(* Logix 5000 project; controller EDS_V35 1769-L16ER-BB1B rev 35.11; software revision 35.00 *)

TASK MainTask (continuous, watchdog 500 ms) : MainProgram

MODULES
   Local : 1769-L16ER-BB1B (PointIO 0, rev 35.11)
      G2410 : vendor 1256 type 43 code 1 (Ethernet 192.168.1.17, rev 6.3, StandardDataDriven RPI 10 ms)
      Discrete_IO : Embedded (PointIO 1, rev 35.11, Output RPI 20 ms)
END_MODULES

PROGRAM MainProgram   (* main routine MainRoutine *)

ROUTINE MainRoutine   (* ladder *)
END_ROUTINE
END_PROGRAM
